// TIA Portal V17 export
// export: Created 2025-03-05T08:00:06.619545Z, ExportSetting WithDefaults, DisplayName Totally Integrated Automation Portal, DisplayVersion V17 Update 8, DisplayName TIA Portal Openness, DisplayVersion V17 Update 8, DisplayName TIA Portal Version Control Interface, DisplayVersion V17, DisplayName SINAMICS Startdrive Advanced, DisplayVersion V17 SP2, DisplayName SINAMICS Startdrive G110M, G120, G120C, G120D, G120P, G115D, DisplayVersion V17 SP2, DisplayName SINAMICS Startdrive G130, G150, S120, S150, SINAMICS MV, S210, DisplayVersion V17 SP2, DisplayName STEP 7 Professional, DisplayVersion V17 Update 8, DisplayName SINUMERIK ONE STEP 7 Toolbox, DisplayVersion V17 Update 12, DisplayName SINUMERIK 840D sl STEP 7 Toolbox, DisplayVersion V17 Update 12, DisplayName STEP 7 Safety, DisplayVersion V17 Update 6, DisplayName WinCC Advanced, DisplayVersion V17 Update 8
FUNCTION "FC2033_RUN_OUT_CYCLE" : Void   // FC2033, LAD
{ S7_Optimized_Access := 'FALSE' }
AUTHOR : ETXETAR
VERSION : 1.0
// stored: AutoNumber false, IsIECCheckEnabled false, SetENOAutomatically false, UDAEnableTagReadback false
   VAR_TEMP
      O_BYTE_0 : Struct   // OPTIONS BYTE 0
         MACH_EMPTY_WITHOUT_STOP_1 : Bool;   // MACHINE EMPTY WITHOUT STOP OPTION
      END_STRUCT;
   END_VAR
   VAR CONSTANT
      FC_NUMBER : DInt := 2033;
   END_VAR
   VAR_TEMP   // added for the SCL form of the ladder/FBD networks
      _w1 : Bool;
      _w2 : Bool;
   END_VAR
BEGIN

REGION Network 1: MACHINE EMPTY WITHOUT STOP OPTION
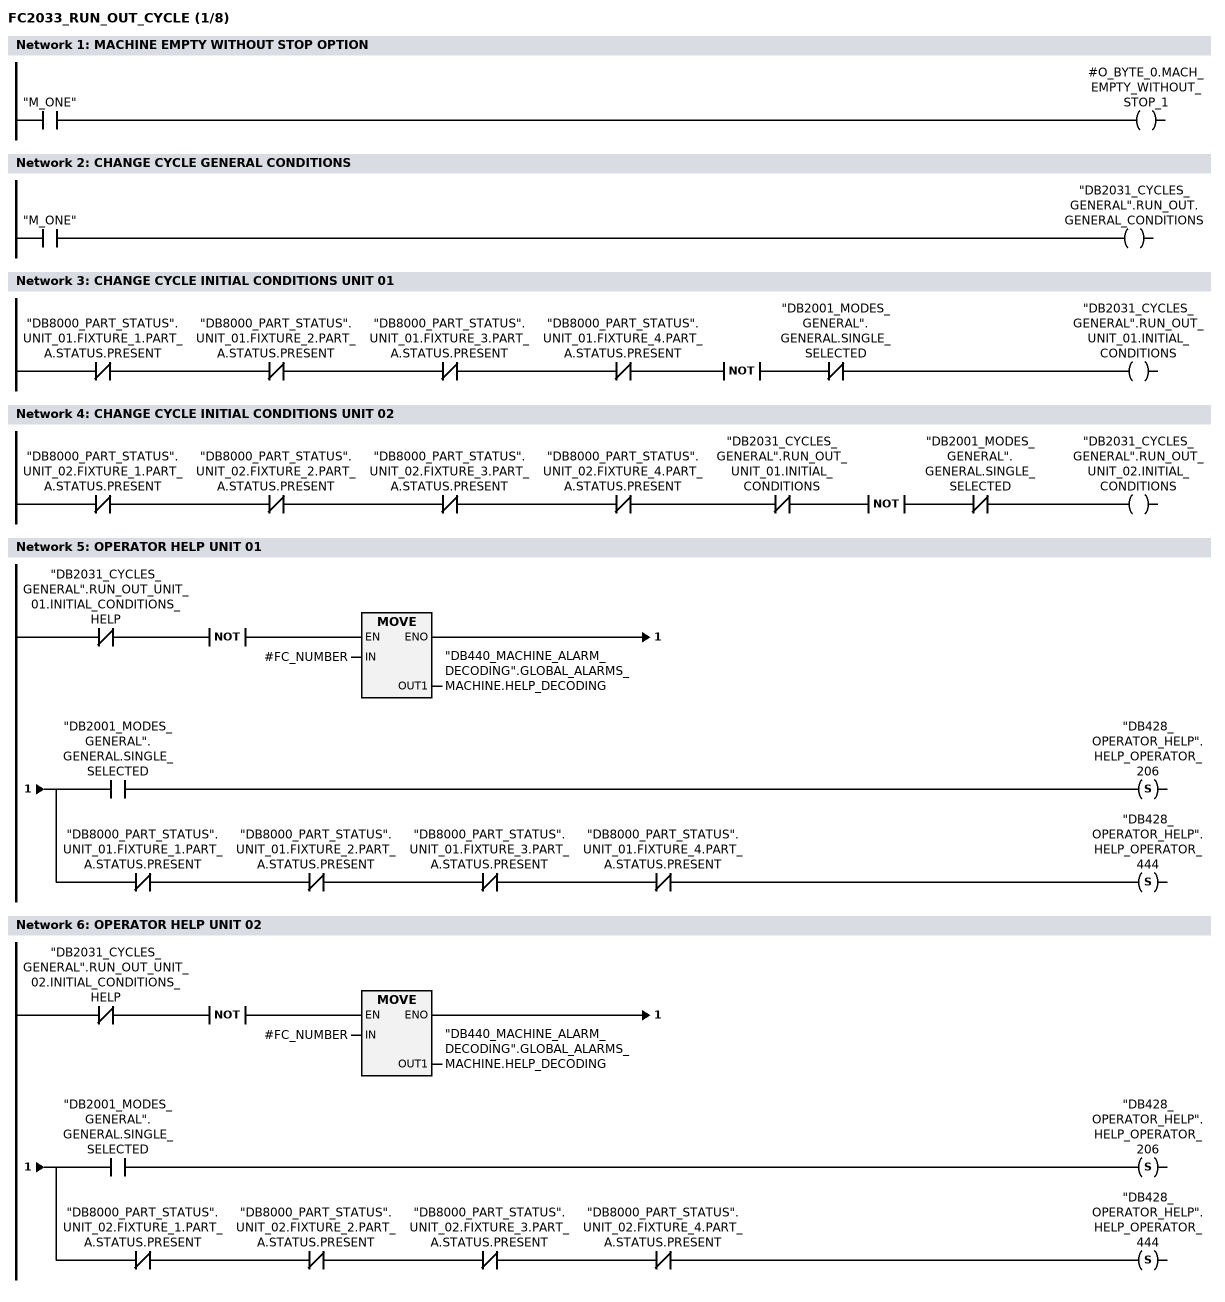
   RUNG wire#powerrail
      Contact( "M_ONE" )
      Coil( #O_BYTE_0.MACH_EMPTY_WITHOUT_STOP_1 )
   END_RUNG
   // the same network as SCL:
   #O_BYTE_0.MACH_EMPTY_WITHOUT_STOP_1 := "M_ONE";
END_REGION

REGION Network 2: CHANGE CYCLE GENERAL CONDITIONS
   RUNG wire#powerrail
      Contact( "M_ONE" )
      Coil( "DB2031_CYCLES_GENERAL".RUN_OUT.GENERAL_CONDITIONS )
   END_RUNG
   // the same network as SCL:
   "DB2031_CYCLES_GENERAL".RUN_OUT.GENERAL_CONDITIONS := "M_ONE";
END_REGION

REGION Network 3: CHANGE CYCLE INITIAL CONDITIONS UNIT 01
   RUNG wire#powerrail
      I_Contact( "DB8000_PART_STATUS".UNIT_01.FIXTURE_1.PART_A.STATUS.PRESENT )
      I_Contact( "DB8000_PART_STATUS".UNIT_01.FIXTURE_2.PART_A.STATUS.PRESENT )
      I_Contact( "DB8000_PART_STATUS".UNIT_01.FIXTURE_3.PART_A.STATUS.PRESENT )
      I_Contact( "DB8000_PART_STATUS".UNIT_01.FIXTURE_4.PART_A.STATUS.PRESENT )
      Not()
      I_Contact( "DB2001_MODES_GENERAL".GENERAL.SINGLE_SELECTED )
      Coil( "DB2031_CYCLES_GENERAL".RUN_OUT_UNIT_01.INITIAL_CONDITIONS )
   END_RUNG
   // the same network as SCL:
   "DB2031_CYCLES_GENERAL".RUN_OUT_UNIT_01.INITIAL_CONDITIONS := NOT (NOT "DB8000_PART_STATUS".UNIT_01.FIXTURE_1.PART_A.STATUS.PRESENT AND NOT "DB8000_PART_STATUS".UNIT_01.FIXTURE_2.PART_A.STATUS.PRESENT AND NOT "DB8000_PART_STATUS".UNIT_01.FIXTURE_3.PART_A.STATUS.PRESENT AND NOT "DB8000_PART_STATUS".UNIT_01.FIXTURE_4.PART_A.STATUS.PRESENT) AND NOT "DB2001_MODES_GENERAL".GENERAL.SINGLE_SELECTED;
END_REGION

REGION Network 4: CHANGE CYCLE INITIAL CONDITIONS UNIT 02
   RUNG wire#powerrail
      I_Contact( "DB8000_PART_STATUS".UNIT_02.FIXTURE_1.PART_A.STATUS.PRESENT )
      I_Contact( "DB8000_PART_STATUS".UNIT_02.FIXTURE_2.PART_A.STATUS.PRESENT )
      I_Contact( "DB8000_PART_STATUS".UNIT_02.FIXTURE_3.PART_A.STATUS.PRESENT )
      I_Contact( "DB8000_PART_STATUS".UNIT_02.FIXTURE_4.PART_A.STATUS.PRESENT )
      I_Contact( "DB2031_CYCLES_GENERAL".RUN_OUT_UNIT_01.INITIAL_CONDITIONS )
      Not()
      I_Contact( "DB2001_MODES_GENERAL".GENERAL.SINGLE_SELECTED )
      Coil( "DB2031_CYCLES_GENERAL".RUN_OUT_UNIT_02.INITIAL_CONDITIONS )
   END_RUNG
   // the same network as SCL:
   "DB2031_CYCLES_GENERAL".RUN_OUT_UNIT_02.INITIAL_CONDITIONS := NOT (NOT "DB8000_PART_STATUS".UNIT_02.FIXTURE_1.PART_A.STATUS.PRESENT AND NOT "DB8000_PART_STATUS".UNIT_02.FIXTURE_2.PART_A.STATUS.PRESENT AND NOT "DB8000_PART_STATUS".UNIT_02.FIXTURE_3.PART_A.STATUS.PRESENT AND NOT "DB8000_PART_STATUS".UNIT_02.FIXTURE_4.PART_A.STATUS.PRESENT AND NOT "DB2031_CYCLES_GENERAL".RUN_OUT_UNIT_01.INITIAL_CONDITIONS) AND NOT "DB2001_MODES_GENERAL".GENERAL.SINGLE_SELECTED;
END_REGION

REGION Network 5: OPERATOR HELP UNIT 01
   RUNG wire#powerrail
      I_Contact( "DB2031_CYCLES_GENERAL".RUN_OUT_UNIT_01.INITIAL_CONDITIONS_HELP )
      Not()
      { S7_GenerateENO := "TRUE" } Move(in := #FC_NUMBER, out1 => "DB440_MACHINE_ALARM_DECODING".GLOBAL_ALARMS_MACHINE.HELP_DECODING)
      wire#w1
      Contact( "DB2001_MODES_GENERAL".GENERAL.SINGLE_SELECTED )
      S_Coil( "DB428_OPERATOR_HELP".HELP_OPERATOR_206 )
   END_RUNG
   RUNG wire#w1
      I_Contact( "DB8000_PART_STATUS".UNIT_01.FIXTURE_1.PART_A.STATUS.PRESENT )
      I_Contact( "DB8000_PART_STATUS".UNIT_01.FIXTURE_2.PART_A.STATUS.PRESENT )
      I_Contact( "DB8000_PART_STATUS".UNIT_01.FIXTURE_3.PART_A.STATUS.PRESENT )
      I_Contact( "DB8000_PART_STATUS".UNIT_01.FIXTURE_4.PART_A.STATUS.PRESENT )
      S_Coil( "DB428_OPERATOR_HELP".HELP_OPERATOR_444 )
   END_RUNG
   // the same network as SCL:
   // ENO of a box is taken as its EN; it also drops when the box reports an error
   #_w1 := NOT (NOT "DB2031_CYCLES_GENERAL".RUN_OUT_UNIT_01.INITIAL_CONDITIONS_HELP);
   IF #_w1 THEN "DB440_MACHINE_ALARM_DECODING".GLOBAL_ALARMS_MACHINE.HELP_DECODING := #FC_NUMBER; END_IF;
   IF #_w1 AND "DB2001_MODES_GENERAL".GENERAL.SINGLE_SELECTED THEN
       "DB428_OPERATOR_HELP".HELP_OPERATOR_206 := TRUE;
   END_IF;
   IF #_w1 AND NOT "DB8000_PART_STATUS".UNIT_01.FIXTURE_1.PART_A.STATUS.PRESENT AND NOT "DB8000_PART_STATUS".UNIT_01.FIXTURE_2.PART_A.STATUS.PRESENT AND NOT "DB8000_PART_STATUS".UNIT_01.FIXTURE_3.PART_A.STATUS.PRESENT AND NOT "DB8000_PART_STATUS".UNIT_01.FIXTURE_4.PART_A.STATUS.PRESENT THEN
       "DB428_OPERATOR_HELP".HELP_OPERATOR_444 := TRUE;
   END_IF;
END_REGION

REGION Network 6: OPERATOR HELP UNIT 02
   RUNG wire#powerrail
      I_Contact( "DB2031_CYCLES_GENERAL".RUN_OUT_UNIT_02.INITIAL_CONDITIONS_HELP )
      Not()
      { S7_GenerateENO := "TRUE" } Move(in := #FC_NUMBER, out1 => "DB440_MACHINE_ALARM_DECODING".GLOBAL_ALARMS_MACHINE.HELP_DECODING)
      wire#w1
      Contact( "DB2001_MODES_GENERAL".GENERAL.SINGLE_SELECTED )
      S_Coil( "DB428_OPERATOR_HELP".HELP_OPERATOR_206 )
   END_RUNG
   RUNG wire#w1
      I_Contact( "DB8000_PART_STATUS".UNIT_02.FIXTURE_1.PART_A.STATUS.PRESENT )
      I_Contact( "DB8000_PART_STATUS".UNIT_02.FIXTURE_2.PART_A.STATUS.PRESENT )
      I_Contact( "DB8000_PART_STATUS".UNIT_02.FIXTURE_3.PART_A.STATUS.PRESENT )
      I_Contact( "DB8000_PART_STATUS".UNIT_02.FIXTURE_4.PART_A.STATUS.PRESENT )
      S_Coil( "DB428_OPERATOR_HELP".HELP_OPERATOR_444 )
   END_RUNG
   // the same network as SCL:
   // ENO of a box is taken as its EN; it also drops when the box reports an error
   #_w1 := NOT (NOT "DB2031_CYCLES_GENERAL".RUN_OUT_UNIT_02.INITIAL_CONDITIONS_HELP);
   IF #_w1 THEN "DB440_MACHINE_ALARM_DECODING".GLOBAL_ALARMS_MACHINE.HELP_DECODING := #FC_NUMBER; END_IF;
   IF #_w1 AND "DB2001_MODES_GENERAL".GENERAL.SINGLE_SELECTED THEN
       "DB428_OPERATOR_HELP".HELP_OPERATOR_206 := TRUE;
   END_IF;
   IF #_w1 AND NOT "DB8000_PART_STATUS".UNIT_02.FIXTURE_1.PART_A.STATUS.PRESENT AND NOT "DB8000_PART_STATUS".UNIT_02.FIXTURE_2.PART_A.STATUS.PRESENT AND NOT "DB8000_PART_STATUS".UNIT_02.FIXTURE_3.PART_A.STATUS.PRESENT AND NOT "DB8000_PART_STATUS".UNIT_02.FIXTURE_4.PART_A.STATUS.PRESENT THEN
       "DB428_OPERATOR_HELP".HELP_OPERATOR_444 := TRUE;
   END_IF;
END_REGION

REGION Network 7: ENABLE REQUEST
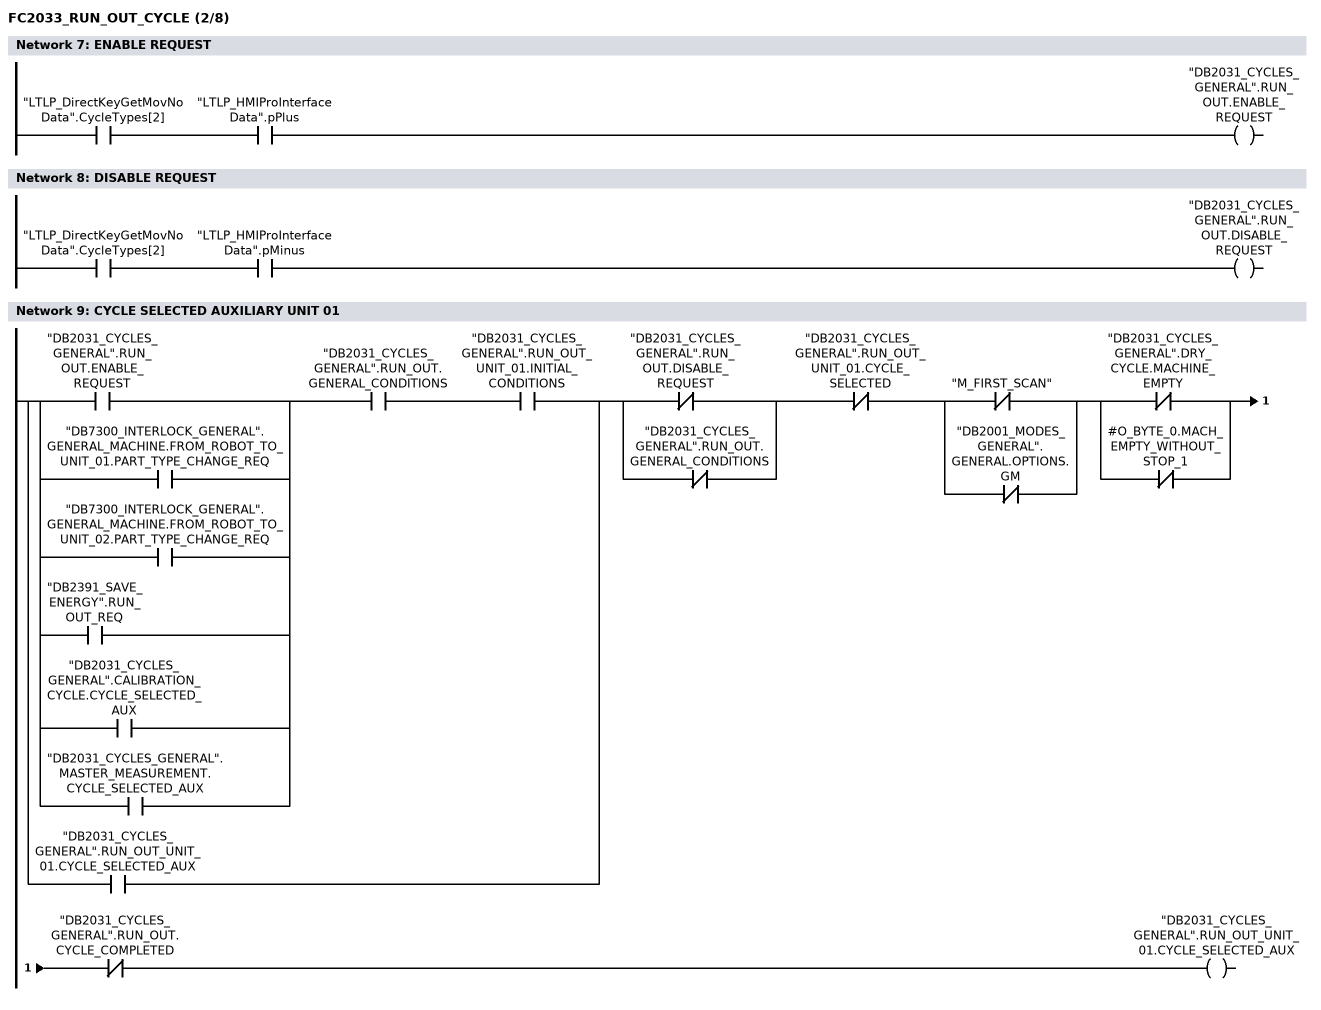
   RUNG wire#powerrail
      Contact( "LTLP_DirectKeyGetMovNoData".CycleTypes[2] )
      Contact( "LTLP_HMIProInterfaceData".pPlus )
      Coil( "DB2031_CYCLES_GENERAL".RUN_OUT.ENABLE_REQUEST )
   END_RUNG
   // the same network as SCL:
   "DB2031_CYCLES_GENERAL".RUN_OUT.ENABLE_REQUEST := "LTLP_DirectKeyGetMovNoData".CycleTypes[2] AND "LTLP_HMIProInterfaceData".pPlus;
END_REGION

REGION Network 8: DISABLE REQUEST
   RUNG wire#powerrail
      Contact( "LTLP_DirectKeyGetMovNoData".CycleTypes[2] )
      Contact( "LTLP_HMIProInterfaceData".pMinus )
      Coil( "DB2031_CYCLES_GENERAL".RUN_OUT.DISABLE_REQUEST )
   END_RUNG
   // the same network as SCL:
   "DB2031_CYCLES_GENERAL".RUN_OUT.DISABLE_REQUEST := "LTLP_DirectKeyGetMovNoData".CycleTypes[2] AND "LTLP_HMIProInterfaceData".pMinus;
END_REGION

REGION Network 9: CYCLE SELECTED AUXILIARY UNIT 01
   RUNG wire#powerrail
      Contact( "DB2031_CYCLES_GENERAL".RUN_OUT.ENABLE_REQUEST )
      wire#w1
      Contact( "DB2031_CYCLES_GENERAL".RUN_OUT.GENERAL_CONDITIONS )
      Contact( "DB2031_CYCLES_GENERAL".RUN_OUT_UNIT_01.INITIAL_CONDITIONS )
      wire#w2
      I_Contact( "DB2031_CYCLES_GENERAL".RUN_OUT.DISABLE_REQUEST )
      wire#w3
      I_Contact( "DB2031_CYCLES_GENERAL".RUN_OUT_UNIT_01.CYCLE_SELECTED )
      wire#w4
      I_Contact( "M_FIRST_SCAN" )
      wire#w5
      I_Contact( "DB2031_CYCLES_GENERAL".DRY_CYCLE.MACHINE_EMPTY )
      wire#w6
      I_Contact( "DB2031_CYCLES_GENERAL".RUN_OUT.CYCLE_COMPLETED )
      Coil( "DB2031_CYCLES_GENERAL".RUN_OUT_UNIT_01.CYCLE_SELECTED_AUX )
   END_RUNG
   RUNG wire#powerrail
      Contact( "DB7300_INTERLOCK_GENERAL".GENERAL_MACHINE.FROM_ROBOT_TO_UNIT_01.PART_TYPE_CHANGE_REQ )
   END_RUNG wire#w1
   RUNG wire#powerrail
      Contact( "DB7300_INTERLOCK_GENERAL".GENERAL_MACHINE.FROM_ROBOT_TO_UNIT_02.PART_TYPE_CHANGE_REQ )
   END_RUNG wire#w1
   RUNG wire#powerrail
      Contact( "DB2391_SAVE_ENERGY".RUN_OUT_REQ )
   END_RUNG wire#w1
   RUNG wire#powerrail
      Contact( "DB2031_CYCLES_GENERAL".CALIBRATION_CYCLE.CYCLE_SELECTED_AUX )
   END_RUNG wire#w1
   RUNG wire#powerrail
      Contact( "DB2031_CYCLES_GENERAL".MASTER_MEASUREMENT.CYCLE_SELECTED_AUX )
   END_RUNG wire#w1
   RUNG wire#powerrail
      Contact( "DB2031_CYCLES_GENERAL".RUN_OUT_UNIT_01.CYCLE_SELECTED_AUX )
   END_RUNG wire#w2
   RUNG wire#w2
      I_Contact( "DB2031_CYCLES_GENERAL".RUN_OUT.GENERAL_CONDITIONS )
   END_RUNG wire#w3
   RUNG wire#w4
      I_Contact( "DB2001_MODES_GENERAL".GENERAL.OPTIONS.GM )
   END_RUNG wire#w5
   RUNG wire#w5
      I_Contact( #O_BYTE_0.MACH_EMPTY_WITHOUT_STOP_1 )
   END_RUNG wire#w6
   // the same network as SCL:
   "DB2031_CYCLES_GENERAL".RUN_OUT_UNIT_01.CYCLE_SELECTED_AUX := ((("DB2031_CYCLES_GENERAL".RUN_OUT.ENABLE_REQUEST OR "DB7300_INTERLOCK_GENERAL".GENERAL_MACHINE.FROM_ROBOT_TO_UNIT_01.PART_TYPE_CHANGE_REQ OR "DB7300_INTERLOCK_GENERAL".GENERAL_MACHINE.FROM_ROBOT_TO_UNIT_02.PART_TYPE_CHANGE_REQ OR "DB2391_SAVE_ENERGY".RUN_OUT_REQ OR "DB2031_CYCLES_GENERAL".CALIBRATION_CYCLE.CYCLE_SELECTED_AUX OR "DB2031_CYCLES_GENERAL".MASTER_MEASUREMENT.CYCLE_SELECTED_AUX) AND "DB2031_CYCLES_GENERAL".RUN_OUT.GENERAL_CONDITIONS AND "DB2031_CYCLES_GENERAL".RUN_OUT_UNIT_01.INITIAL_CONDITIONS) OR "DB2031_CYCLES_GENERAL".RUN_OUT_UNIT_01.CYCLE_SELECTED_AUX) AND (NOT "DB2031_CYCLES_GENERAL".RUN_OUT.DISABLE_REQUEST OR NOT "DB2031_CYCLES_GENERAL".RUN_OUT.GENERAL_CONDITIONS) AND NOT "DB2031_CYCLES_GENERAL".RUN_OUT_UNIT_01.CYCLE_SELECTED AND (NOT "M_FIRST_SCAN" OR NOT "DB2001_MODES_GENERAL".GENERAL.OPTIONS.GM) AND (NOT "DB2031_CYCLES_GENERAL".DRY_CYCLE.MACHINE_EMPTY OR NOT #O_BYTE_0.MACH_EMPTY_WITHOUT_STOP_1) AND NOT "DB2031_CYCLES_GENERAL".RUN_OUT.CYCLE_COMPLETED;
END_REGION

REGION Network 10: CYCLE SELECTED AUXILIARY UNIT 02
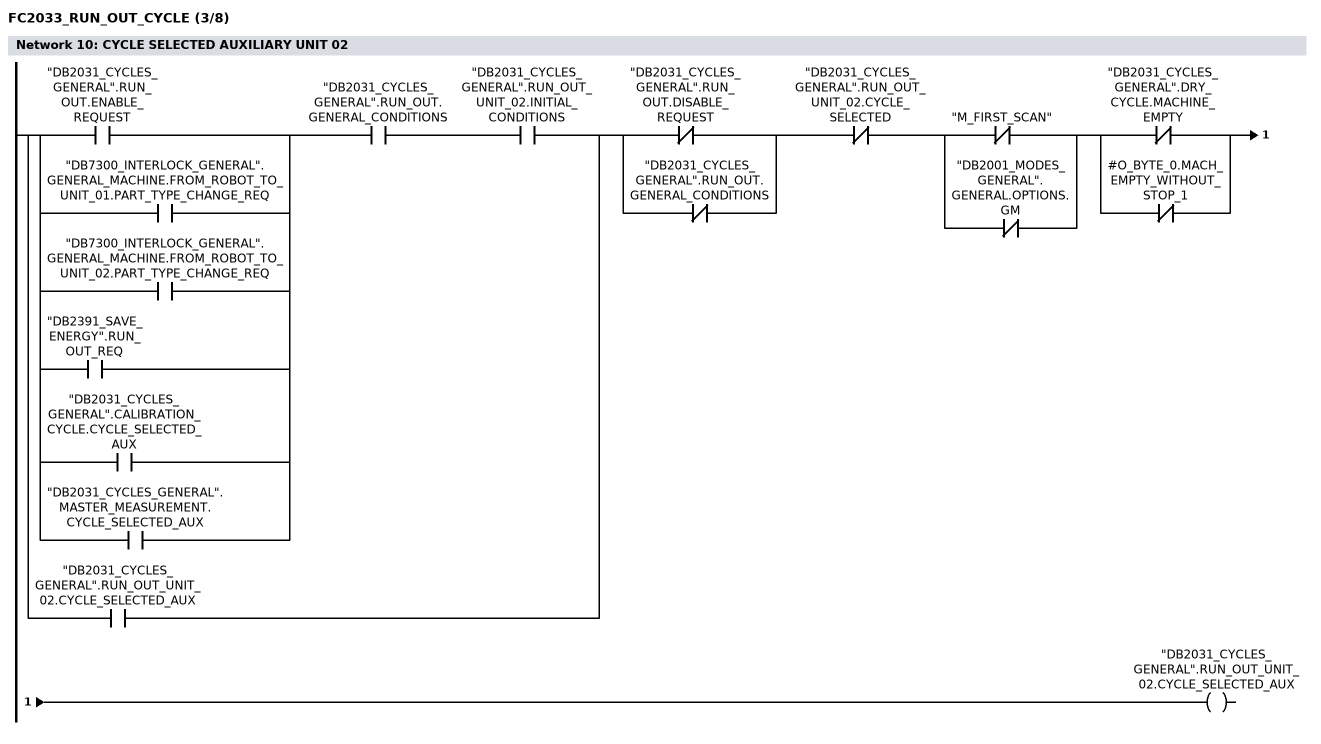
   RUNG wire#powerrail
      Contact( "DB2031_CYCLES_GENERAL".RUN_OUT.ENABLE_REQUEST )
      wire#w1
      Contact( "DB2031_CYCLES_GENERAL".RUN_OUT.GENERAL_CONDITIONS )
      Contact( "DB2031_CYCLES_GENERAL".RUN_OUT_UNIT_02.INITIAL_CONDITIONS )
      wire#w2
      I_Contact( "DB2031_CYCLES_GENERAL".RUN_OUT.DISABLE_REQUEST )
      wire#w3
      I_Contact( "DB2031_CYCLES_GENERAL".RUN_OUT_UNIT_02.CYCLE_SELECTED )
      wire#w4
      I_Contact( "M_FIRST_SCAN" )
      wire#w5
      I_Contact( "DB2031_CYCLES_GENERAL".DRY_CYCLE.MACHINE_EMPTY )
      wire#w6
      Coil( "DB2031_CYCLES_GENERAL".RUN_OUT_UNIT_02.CYCLE_SELECTED_AUX )
   END_RUNG
   RUNG wire#powerrail
      Contact( "DB7300_INTERLOCK_GENERAL".GENERAL_MACHINE.FROM_ROBOT_TO_UNIT_01.PART_TYPE_CHANGE_REQ )
   END_RUNG wire#w1
   RUNG wire#powerrail
      Contact( "DB7300_INTERLOCK_GENERAL".GENERAL_MACHINE.FROM_ROBOT_TO_UNIT_02.PART_TYPE_CHANGE_REQ )
   END_RUNG wire#w1
   RUNG wire#powerrail
      Contact( "DB2391_SAVE_ENERGY".RUN_OUT_REQ )
   END_RUNG wire#w1
   RUNG wire#powerrail
      Contact( "DB2031_CYCLES_GENERAL".CALIBRATION_CYCLE.CYCLE_SELECTED_AUX )
   END_RUNG wire#w1
   RUNG wire#powerrail
      Contact( "DB2031_CYCLES_GENERAL".MASTER_MEASUREMENT.CYCLE_SELECTED_AUX )
   END_RUNG wire#w1
   RUNG wire#powerrail
      Contact( "DB2031_CYCLES_GENERAL".RUN_OUT_UNIT_02.CYCLE_SELECTED_AUX )
   END_RUNG wire#w2
   RUNG wire#w2
      I_Contact( "DB2031_CYCLES_GENERAL".RUN_OUT.GENERAL_CONDITIONS )
   END_RUNG wire#w3
   RUNG wire#w4
      I_Contact( "DB2001_MODES_GENERAL".GENERAL.OPTIONS.GM )
   END_RUNG wire#w5
   RUNG wire#w5
      I_Contact( #O_BYTE_0.MACH_EMPTY_WITHOUT_STOP_1 )
   END_RUNG wire#w6
   // the same network as SCL:
   "DB2031_CYCLES_GENERAL".RUN_OUT_UNIT_02.CYCLE_SELECTED_AUX := ((("DB2031_CYCLES_GENERAL".RUN_OUT.ENABLE_REQUEST OR "DB7300_INTERLOCK_GENERAL".GENERAL_MACHINE.FROM_ROBOT_TO_UNIT_01.PART_TYPE_CHANGE_REQ OR "DB7300_INTERLOCK_GENERAL".GENERAL_MACHINE.FROM_ROBOT_TO_UNIT_02.PART_TYPE_CHANGE_REQ OR "DB2391_SAVE_ENERGY".RUN_OUT_REQ OR "DB2031_CYCLES_GENERAL".CALIBRATION_CYCLE.CYCLE_SELECTED_AUX OR "DB2031_CYCLES_GENERAL".MASTER_MEASUREMENT.CYCLE_SELECTED_AUX) AND "DB2031_CYCLES_GENERAL".RUN_OUT.GENERAL_CONDITIONS AND "DB2031_CYCLES_GENERAL".RUN_OUT_UNIT_02.INITIAL_CONDITIONS) OR "DB2031_CYCLES_GENERAL".RUN_OUT_UNIT_02.CYCLE_SELECTED_AUX) AND (NOT "DB2031_CYCLES_GENERAL".RUN_OUT.DISABLE_REQUEST OR NOT "DB2031_CYCLES_GENERAL".RUN_OUT.GENERAL_CONDITIONS) AND NOT "DB2031_CYCLES_GENERAL".RUN_OUT_UNIT_02.CYCLE_SELECTED AND (NOT "M_FIRST_SCAN" OR NOT "DB2001_MODES_GENERAL".GENERAL.OPTIONS.GM) AND (NOT "DB2031_CYCLES_GENERAL".DRY_CYCLE.MACHINE_EMPTY OR NOT #O_BYTE_0.MACH_EMPTY_WITHOUT_STOP_1);
END_REGION

REGION Network 11: CYCLE SELECTED UNIT 01
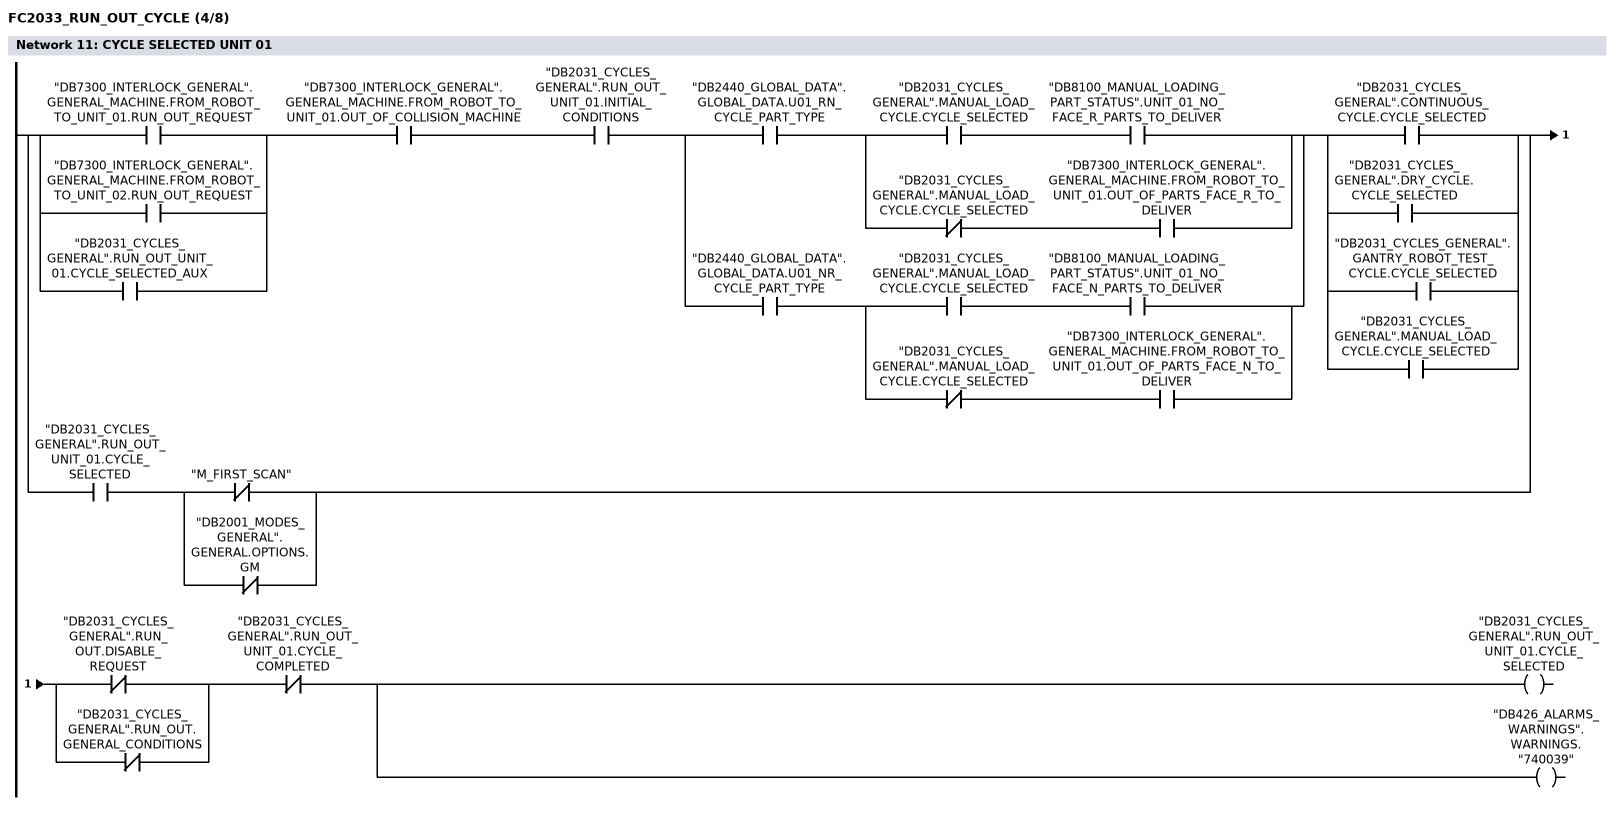
   RUNG wire#powerrail
      Contact( "DB7300_INTERLOCK_GENERAL".GENERAL_MACHINE.FROM_ROBOT_TO_UNIT_01.RUN_OUT_REQUEST )
      wire#w1
      Contact( "DB7300_INTERLOCK_GENERAL".GENERAL_MACHINE.FROM_ROBOT_TO_UNIT_01.OUT_OF_COLLISION_MACHINE )
      Contact( "DB2031_CYCLES_GENERAL".RUN_OUT_UNIT_01.INITIAL_CONDITIONS )
      wire#w2
      Contact( "DB2440_GLOBAL_DATA".GLOBAL_DATA.U01_RN_CYCLE_PART_TYPE )
      wire#w3
      Contact( "DB2031_CYCLES_GENERAL".MANUAL_LOAD_CYCLE.CYCLE_SELECTED )
      Contact( "DB8100_MANUAL_LOADING_PART_STATUS".UNIT_01_NO_FACE_R_PARTS_TO_DELIVER )
      wire#w4
      Contact( "DB2031_CYCLES_GENERAL".CONTINUOUS_CYCLE.CYCLE_SELECTED )
      wire#w6
      I_Contact( "DB2031_CYCLES_GENERAL".RUN_OUT.DISABLE_REQUEST )
      wire#w8
      I_Contact( "DB2031_CYCLES_GENERAL".RUN_OUT_UNIT_01.CYCLE_COMPLETED )
      wire#w9
      Coil( "DB2031_CYCLES_GENERAL".RUN_OUT_UNIT_01.CYCLE_SELECTED )
   END_RUNG
   RUNG wire#powerrail
      Contact( "DB7300_INTERLOCK_GENERAL".GENERAL_MACHINE.FROM_ROBOT_TO_UNIT_02.RUN_OUT_REQUEST )
   END_RUNG wire#w1
   RUNG wire#powerrail
      Contact( "DB2031_CYCLES_GENERAL".RUN_OUT_UNIT_01.CYCLE_SELECTED_AUX )
   END_RUNG wire#w1
   RUNG wire#w3
      I_Contact( "DB2031_CYCLES_GENERAL".MANUAL_LOAD_CYCLE.CYCLE_SELECTED )
      Contact( "DB7300_INTERLOCK_GENERAL".GENERAL_MACHINE.FROM_ROBOT_TO_UNIT_01.OUT_OF_PARTS_FACE_R_TO_DELIVER )
   END_RUNG wire#w4
   RUNG wire#w2
      Contact( "DB2440_GLOBAL_DATA".GLOBAL_DATA.U01_NR_CYCLE_PART_TYPE )
      wire#w5
      Contact( "DB2031_CYCLES_GENERAL".MANUAL_LOAD_CYCLE.CYCLE_SELECTED )
      Contact( "DB8100_MANUAL_LOADING_PART_STATUS".UNIT_01_NO_FACE_N_PARTS_TO_DELIVER )
   END_RUNG wire#w4
   RUNG wire#w5
      I_Contact( "DB2031_CYCLES_GENERAL".MANUAL_LOAD_CYCLE.CYCLE_SELECTED )
      Contact( "DB7300_INTERLOCK_GENERAL".GENERAL_MACHINE.FROM_ROBOT_TO_UNIT_01.OUT_OF_PARTS_FACE_N_TO_DELIVER )
   END_RUNG wire#w4
   RUNG wire#w4
      Contact( "DB2031_CYCLES_GENERAL".DRY_CYCLE.CYCLE_SELECTED )
   END_RUNG wire#w6
   RUNG wire#w4
      Contact( "DB2031_CYCLES_GENERAL".GANTRY_ROBOT_TEST_CYCLE.CYCLE_SELECTED )
   END_RUNG wire#w6
   RUNG wire#w4
      Contact( "DB2031_CYCLES_GENERAL".MANUAL_LOAD_CYCLE.CYCLE_SELECTED )
   END_RUNG wire#w6
   RUNG wire#powerrail
      Contact( "DB2031_CYCLES_GENERAL".RUN_OUT_UNIT_01.CYCLE_SELECTED )
      wire#w7
      I_Contact( "M_FIRST_SCAN" )
   END_RUNG wire#w6
   RUNG wire#w7
      I_Contact( "DB2001_MODES_GENERAL".GENERAL.OPTIONS.GM )
   END_RUNG wire#w6
   RUNG wire#w6
      I_Contact( "DB2031_CYCLES_GENERAL".RUN_OUT.GENERAL_CONDITIONS )
   END_RUNG wire#w8
   RUNG wire#w9
      Coil( "DB426_ALARMS_WARNINGS".WARNINGS."740039" )
   END_RUNG
   // the same network as SCL:
   "DB2031_CYCLES_GENERAL".RUN_OUT_UNIT_01.CYCLE_SELECTED := ((("DB7300_INTERLOCK_GENERAL".GENERAL_MACHINE.FROM_ROBOT_TO_UNIT_01.RUN_OUT_REQUEST OR "DB7300_INTERLOCK_GENERAL".GENERAL_MACHINE.FROM_ROBOT_TO_UNIT_02.RUN_OUT_REQUEST OR "DB2031_CYCLES_GENERAL".RUN_OUT_UNIT_01.CYCLE_SELECTED_AUX) AND "DB7300_INTERLOCK_GENERAL".GENERAL_MACHINE.FROM_ROBOT_TO_UNIT_01.OUT_OF_COLLISION_MACHINE AND "DB2031_CYCLES_GENERAL".RUN_OUT_UNIT_01.INITIAL_CONDITIONS AND (("DB2440_GLOBAL_DATA".GLOBAL_DATA.U01_RN_CYCLE_PART_TYPE AND (("DB2031_CYCLES_GENERAL".MANUAL_LOAD_CYCLE.CYCLE_SELECTED AND "DB8100_MANUAL_LOADING_PART_STATUS".UNIT_01_NO_FACE_R_PARTS_TO_DELIVER) OR (NOT "DB2031_CYCLES_GENERAL".MANUAL_LOAD_CYCLE.CYCLE_SELECTED AND "DB7300_INTERLOCK_GENERAL".GENERAL_MACHINE.FROM_ROBOT_TO_UNIT_01.OUT_OF_PARTS_FACE_R_TO_DELIVER))) OR ("DB2440_GLOBAL_DATA".GLOBAL_DATA.U01_NR_CYCLE_PART_TYPE AND (("DB2031_CYCLES_GENERAL".MANUAL_LOAD_CYCLE.CYCLE_SELECTED AND "DB8100_MANUAL_LOADING_PART_STATUS".UNIT_01_NO_FACE_N_PARTS_TO_DELIVER) OR (NOT "DB2031_CYCLES_GENERAL".MANUAL_LOAD_CYCLE.CYCLE_SELECTED AND "DB7300_INTERLOCK_GENERAL".GENERAL_MACHINE.FROM_ROBOT_TO_UNIT_01.OUT_OF_PARTS_FACE_N_TO_DELIVER)))) AND ("DB2031_CYCLES_GENERAL".CONTINUOUS_CYCLE.CYCLE_SELECTED OR "DB2031_CYCLES_GENERAL".DRY_CYCLE.CYCLE_SELECTED OR "DB2031_CYCLES_GENERAL".GANTRY_ROBOT_TEST_CYCLE.CYCLE_SELECTED OR "DB2031_CYCLES_GENERAL".MANUAL_LOAD_CYCLE.CYCLE_SELECTED)) OR ("DB2031_CYCLES_GENERAL".RUN_OUT_UNIT_01.CYCLE_SELECTED AND (NOT "M_FIRST_SCAN" OR NOT "DB2001_MODES_GENERAL".GENERAL.OPTIONS.GM))) AND (NOT "DB2031_CYCLES_GENERAL".RUN_OUT.DISABLE_REQUEST OR NOT "DB2031_CYCLES_GENERAL".RUN_OUT.GENERAL_CONDITIONS) AND NOT "DB2031_CYCLES_GENERAL".RUN_OUT_UNIT_01.CYCLE_COMPLETED;
   "DB426_ALARMS_WARNINGS".WARNINGS."740039" := "DB2031_CYCLES_GENERAL".RUN_OUT_UNIT_01.CYCLE_SELECTED;
END_REGION

REGION Network 12: CYCLE SELECTED UNIT 02
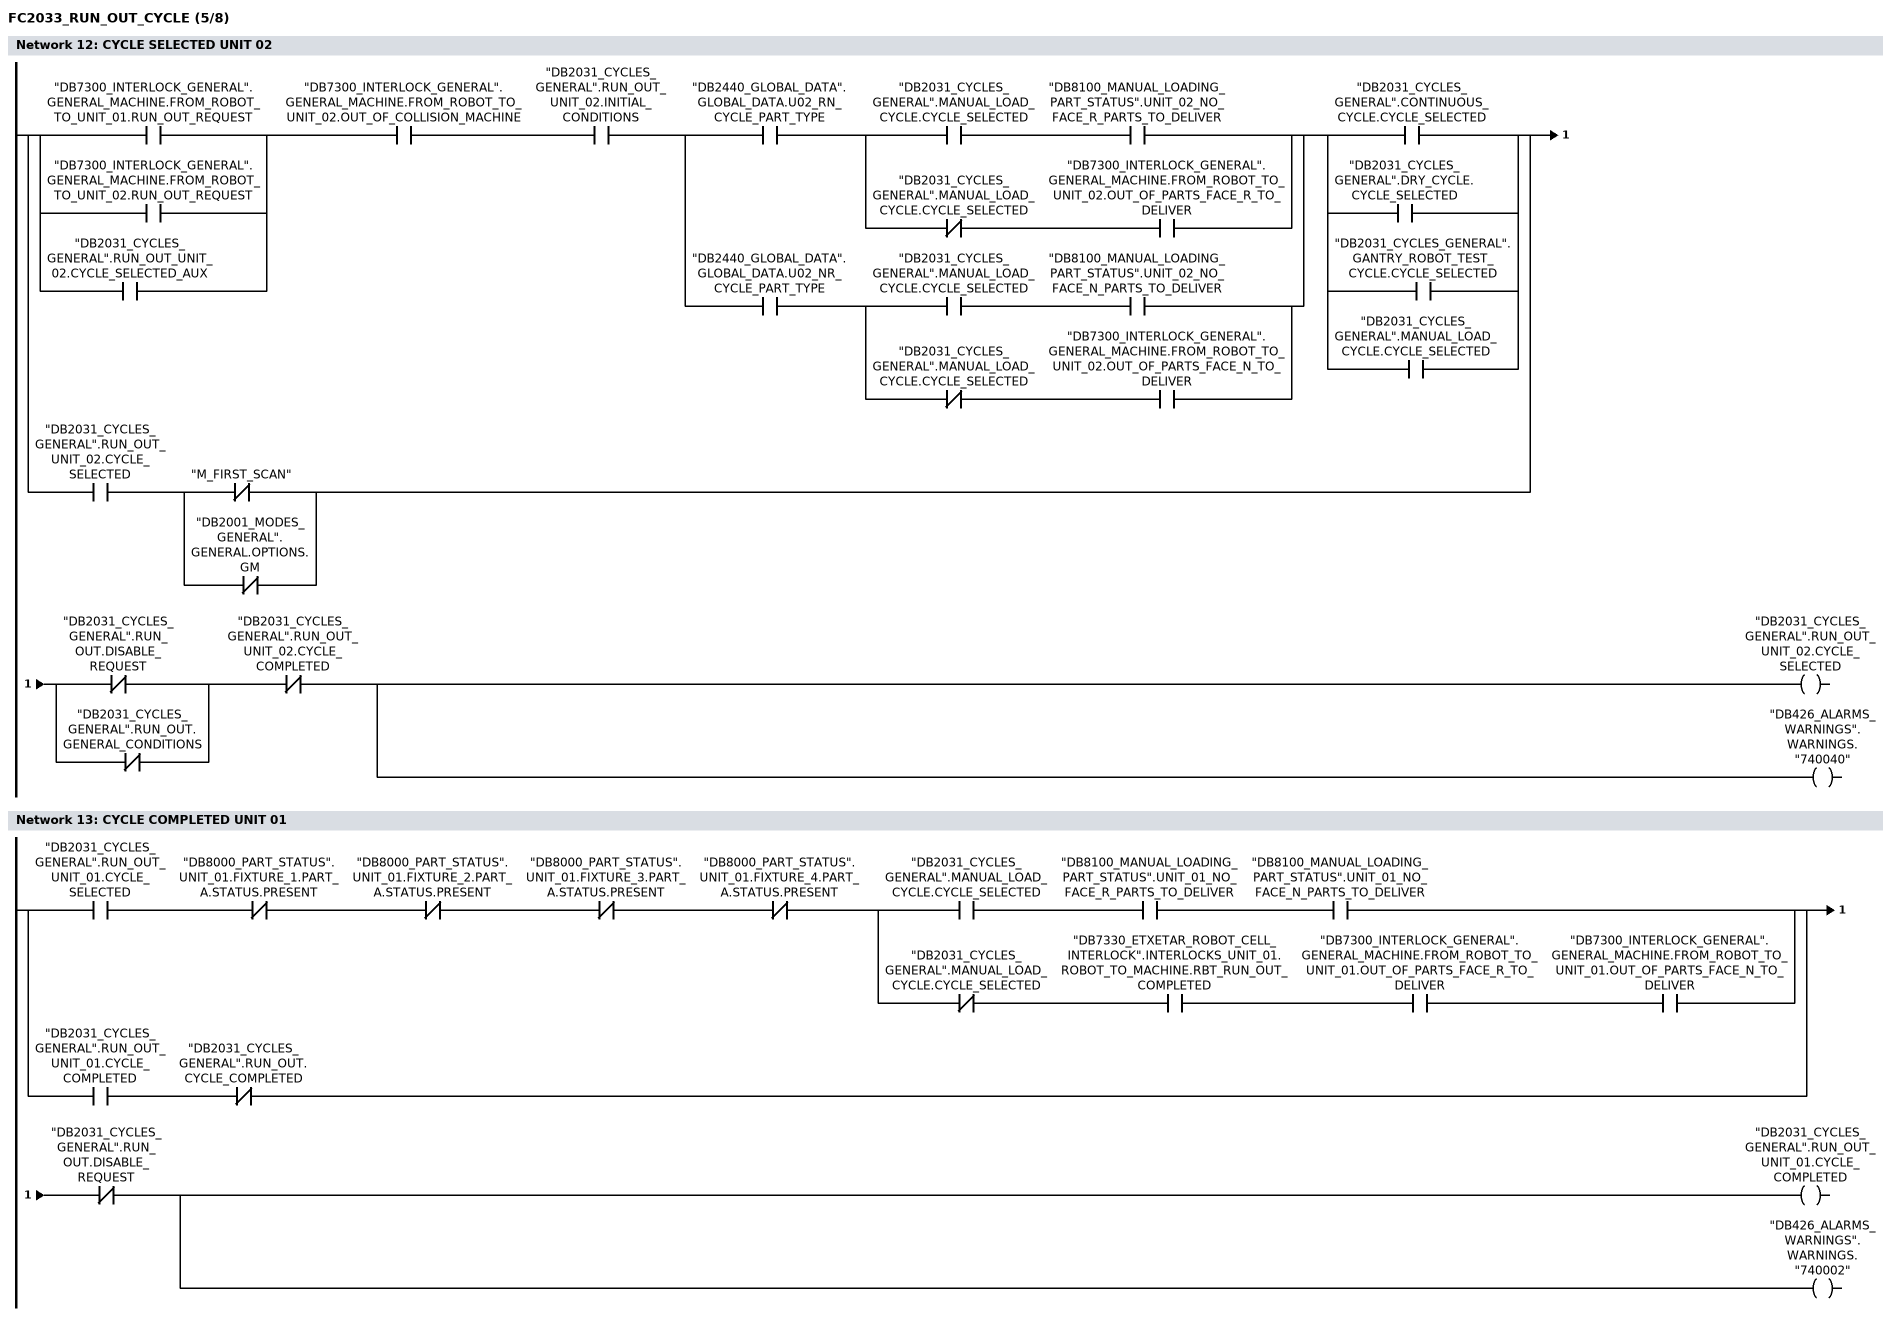
   RUNG wire#powerrail
      Contact( "DB7300_INTERLOCK_GENERAL".GENERAL_MACHINE.FROM_ROBOT_TO_UNIT_01.RUN_OUT_REQUEST )
      wire#w1
      Contact( "DB7300_INTERLOCK_GENERAL".GENERAL_MACHINE.FROM_ROBOT_TO_UNIT_02.OUT_OF_COLLISION_MACHINE )
      Contact( "DB2031_CYCLES_GENERAL".RUN_OUT_UNIT_02.INITIAL_CONDITIONS )
      wire#w2
      Contact( "DB2440_GLOBAL_DATA".GLOBAL_DATA.U02_RN_CYCLE_PART_TYPE )
      wire#w3
      Contact( "DB2031_CYCLES_GENERAL".MANUAL_LOAD_CYCLE.CYCLE_SELECTED )
      Contact( "DB8100_MANUAL_LOADING_PART_STATUS".UNIT_02_NO_FACE_R_PARTS_TO_DELIVER )
      wire#w4
      Contact( "DB2031_CYCLES_GENERAL".CONTINUOUS_CYCLE.CYCLE_SELECTED )
      wire#w6
      I_Contact( "DB2031_CYCLES_GENERAL".RUN_OUT.DISABLE_REQUEST )
      wire#w8
      I_Contact( "DB2031_CYCLES_GENERAL".RUN_OUT_UNIT_02.CYCLE_COMPLETED )
      wire#w9
      Coil( "DB2031_CYCLES_GENERAL".RUN_OUT_UNIT_02.CYCLE_SELECTED )
   END_RUNG
   RUNG wire#powerrail
      Contact( "DB7300_INTERLOCK_GENERAL".GENERAL_MACHINE.FROM_ROBOT_TO_UNIT_02.RUN_OUT_REQUEST )
   END_RUNG wire#w1
   RUNG wire#powerrail
      Contact( "DB2031_CYCLES_GENERAL".RUN_OUT_UNIT_02.CYCLE_SELECTED_AUX )
   END_RUNG wire#w1
   RUNG wire#w3
      I_Contact( "DB2031_CYCLES_GENERAL".MANUAL_LOAD_CYCLE.CYCLE_SELECTED )
      Contact( "DB7300_INTERLOCK_GENERAL".GENERAL_MACHINE.FROM_ROBOT_TO_UNIT_02.OUT_OF_PARTS_FACE_R_TO_DELIVER )
   END_RUNG wire#w4
   RUNG wire#w2
      Contact( "DB2440_GLOBAL_DATA".GLOBAL_DATA.U02_NR_CYCLE_PART_TYPE )
      wire#w5
      Contact( "DB2031_CYCLES_GENERAL".MANUAL_LOAD_CYCLE.CYCLE_SELECTED )
      Contact( "DB8100_MANUAL_LOADING_PART_STATUS".UNIT_02_NO_FACE_N_PARTS_TO_DELIVER )
   END_RUNG wire#w4
   RUNG wire#w5
      I_Contact( "DB2031_CYCLES_GENERAL".MANUAL_LOAD_CYCLE.CYCLE_SELECTED )
      Contact( "DB7300_INTERLOCK_GENERAL".GENERAL_MACHINE.FROM_ROBOT_TO_UNIT_02.OUT_OF_PARTS_FACE_N_TO_DELIVER )
   END_RUNG wire#w4
   RUNG wire#w4
      Contact( "DB2031_CYCLES_GENERAL".DRY_CYCLE.CYCLE_SELECTED )
   END_RUNG wire#w6
   RUNG wire#w4
      Contact( "DB2031_CYCLES_GENERAL".GANTRY_ROBOT_TEST_CYCLE.CYCLE_SELECTED )
   END_RUNG wire#w6
   RUNG wire#w4
      Contact( "DB2031_CYCLES_GENERAL".MANUAL_LOAD_CYCLE.CYCLE_SELECTED )
   END_RUNG wire#w6
   RUNG wire#powerrail
      Contact( "DB2031_CYCLES_GENERAL".RUN_OUT_UNIT_02.CYCLE_SELECTED )
      wire#w7
      I_Contact( "M_FIRST_SCAN" )
   END_RUNG wire#w6
   RUNG wire#w7
      I_Contact( "DB2001_MODES_GENERAL".GENERAL.OPTIONS.GM )
   END_RUNG wire#w6
   RUNG wire#w6
      I_Contact( "DB2031_CYCLES_GENERAL".RUN_OUT.GENERAL_CONDITIONS )
   END_RUNG wire#w8
   RUNG wire#w9
      Coil( "DB426_ALARMS_WARNINGS".WARNINGS."740040" )
   END_RUNG
   // the same network as SCL:
   "DB2031_CYCLES_GENERAL".RUN_OUT_UNIT_02.CYCLE_SELECTED := ((("DB7300_INTERLOCK_GENERAL".GENERAL_MACHINE.FROM_ROBOT_TO_UNIT_01.RUN_OUT_REQUEST OR "DB7300_INTERLOCK_GENERAL".GENERAL_MACHINE.FROM_ROBOT_TO_UNIT_02.RUN_OUT_REQUEST OR "DB2031_CYCLES_GENERAL".RUN_OUT_UNIT_02.CYCLE_SELECTED_AUX) AND "DB7300_INTERLOCK_GENERAL".GENERAL_MACHINE.FROM_ROBOT_TO_UNIT_02.OUT_OF_COLLISION_MACHINE AND "DB2031_CYCLES_GENERAL".RUN_OUT_UNIT_02.INITIAL_CONDITIONS AND (("DB2440_GLOBAL_DATA".GLOBAL_DATA.U02_RN_CYCLE_PART_TYPE AND (("DB2031_CYCLES_GENERAL".MANUAL_LOAD_CYCLE.CYCLE_SELECTED AND "DB8100_MANUAL_LOADING_PART_STATUS".UNIT_02_NO_FACE_R_PARTS_TO_DELIVER) OR (NOT "DB2031_CYCLES_GENERAL".MANUAL_LOAD_CYCLE.CYCLE_SELECTED AND "DB7300_INTERLOCK_GENERAL".GENERAL_MACHINE.FROM_ROBOT_TO_UNIT_02.OUT_OF_PARTS_FACE_R_TO_DELIVER))) OR ("DB2440_GLOBAL_DATA".GLOBAL_DATA.U02_NR_CYCLE_PART_TYPE AND (("DB2031_CYCLES_GENERAL".MANUAL_LOAD_CYCLE.CYCLE_SELECTED AND "DB8100_MANUAL_LOADING_PART_STATUS".UNIT_02_NO_FACE_N_PARTS_TO_DELIVER) OR (NOT "DB2031_CYCLES_GENERAL".MANUAL_LOAD_CYCLE.CYCLE_SELECTED AND "DB7300_INTERLOCK_GENERAL".GENERAL_MACHINE.FROM_ROBOT_TO_UNIT_02.OUT_OF_PARTS_FACE_N_TO_DELIVER)))) AND ("DB2031_CYCLES_GENERAL".CONTINUOUS_CYCLE.CYCLE_SELECTED OR "DB2031_CYCLES_GENERAL".DRY_CYCLE.CYCLE_SELECTED OR "DB2031_CYCLES_GENERAL".GANTRY_ROBOT_TEST_CYCLE.CYCLE_SELECTED OR "DB2031_CYCLES_GENERAL".MANUAL_LOAD_CYCLE.CYCLE_SELECTED)) OR ("DB2031_CYCLES_GENERAL".RUN_OUT_UNIT_02.CYCLE_SELECTED AND (NOT "M_FIRST_SCAN" OR NOT "DB2001_MODES_GENERAL".GENERAL.OPTIONS.GM))) AND (NOT "DB2031_CYCLES_GENERAL".RUN_OUT.DISABLE_REQUEST OR NOT "DB2031_CYCLES_GENERAL".RUN_OUT.GENERAL_CONDITIONS) AND NOT "DB2031_CYCLES_GENERAL".RUN_OUT_UNIT_02.CYCLE_COMPLETED;
   "DB426_ALARMS_WARNINGS".WARNINGS."740040" := "DB2031_CYCLES_GENERAL".RUN_OUT_UNIT_02.CYCLE_SELECTED;
END_REGION

REGION Network 13: CYCLE COMPLETED UNIT 01
   RUNG wire#powerrail
      Contact( "DB2031_CYCLES_GENERAL".RUN_OUT_UNIT_01.CYCLE_SELECTED )
      I_Contact( "DB8000_PART_STATUS".UNIT_01.FIXTURE_1.PART_A.STATUS.PRESENT )
      I_Contact( "DB8000_PART_STATUS".UNIT_01.FIXTURE_2.PART_A.STATUS.PRESENT )
      I_Contact( "DB8000_PART_STATUS".UNIT_01.FIXTURE_3.PART_A.STATUS.PRESENT )
      I_Contact( "DB8000_PART_STATUS".UNIT_01.FIXTURE_4.PART_A.STATUS.PRESENT )
      wire#w1
      Contact( "DB2031_CYCLES_GENERAL".MANUAL_LOAD_CYCLE.CYCLE_SELECTED )
      Contact( "DB8100_MANUAL_LOADING_PART_STATUS".UNIT_01_NO_FACE_R_PARTS_TO_DELIVER )
      Contact( "DB8100_MANUAL_LOADING_PART_STATUS".UNIT_01_NO_FACE_N_PARTS_TO_DELIVER )
      wire#w2
      I_Contact( "DB2031_CYCLES_GENERAL".RUN_OUT.DISABLE_REQUEST )
      wire#w3
      Coil( "DB2031_CYCLES_GENERAL".RUN_OUT_UNIT_01.CYCLE_COMPLETED )
   END_RUNG
   RUNG wire#w1
      I_Contact( "DB2031_CYCLES_GENERAL".MANUAL_LOAD_CYCLE.CYCLE_SELECTED )
      Contact( "DB7330_ETXETAR_ROBOT_CELL_INTERLOCK".INTERLOCKS_UNIT_01.ROBOT_TO_MACHINE.RBT_RUN_OUT_COMPLETED )
      Contact( "DB7300_INTERLOCK_GENERAL".GENERAL_MACHINE.FROM_ROBOT_TO_UNIT_01.OUT_OF_PARTS_FACE_R_TO_DELIVER )
      Contact( "DB7300_INTERLOCK_GENERAL".GENERAL_MACHINE.FROM_ROBOT_TO_UNIT_01.OUT_OF_PARTS_FACE_N_TO_DELIVER )
   END_RUNG wire#w2
   RUNG wire#powerrail
      Contact( "DB2031_CYCLES_GENERAL".RUN_OUT_UNIT_01.CYCLE_COMPLETED )
      I_Contact( "DB2031_CYCLES_GENERAL".RUN_OUT.CYCLE_COMPLETED )
   END_RUNG wire#w2
   RUNG wire#w3
      Coil( "DB426_ALARMS_WARNINGS".WARNINGS."740002" )
   END_RUNG
   // the same network as SCL:
   "DB2031_CYCLES_GENERAL".RUN_OUT_UNIT_01.CYCLE_COMPLETED := (("DB2031_CYCLES_GENERAL".RUN_OUT_UNIT_01.CYCLE_SELECTED AND NOT "DB8000_PART_STATUS".UNIT_01.FIXTURE_1.PART_A.STATUS.PRESENT AND NOT "DB8000_PART_STATUS".UNIT_01.FIXTURE_2.PART_A.STATUS.PRESENT AND NOT "DB8000_PART_STATUS".UNIT_01.FIXTURE_3.PART_A.STATUS.PRESENT AND NOT "DB8000_PART_STATUS".UNIT_01.FIXTURE_4.PART_A.STATUS.PRESENT AND (("DB2031_CYCLES_GENERAL".MANUAL_LOAD_CYCLE.CYCLE_SELECTED AND "DB8100_MANUAL_LOADING_PART_STATUS".UNIT_01_NO_FACE_R_PARTS_TO_DELIVER AND "DB8100_MANUAL_LOADING_PART_STATUS".UNIT_01_NO_FACE_N_PARTS_TO_DELIVER) OR (NOT "DB2031_CYCLES_GENERAL".MANUAL_LOAD_CYCLE.CYCLE_SELECTED AND "DB7330_ETXETAR_ROBOT_CELL_INTERLOCK".INTERLOCKS_UNIT_01.ROBOT_TO_MACHINE.RBT_RUN_OUT_COMPLETED AND "DB7300_INTERLOCK_GENERAL".GENERAL_MACHINE.FROM_ROBOT_TO_UNIT_01.OUT_OF_PARTS_FACE_R_TO_DELIVER AND "DB7300_INTERLOCK_GENERAL".GENERAL_MACHINE.FROM_ROBOT_TO_UNIT_01.OUT_OF_PARTS_FACE_N_TO_DELIVER))) OR ("DB2031_CYCLES_GENERAL".RUN_OUT_UNIT_01.CYCLE_COMPLETED AND NOT "DB2031_CYCLES_GENERAL".RUN_OUT.CYCLE_COMPLETED)) AND NOT "DB2031_CYCLES_GENERAL".RUN_OUT.DISABLE_REQUEST;
   "DB426_ALARMS_WARNINGS".WARNINGS."740002" := "DB2031_CYCLES_GENERAL".RUN_OUT_UNIT_01.CYCLE_COMPLETED;
END_REGION

REGION Network 14: CYCLE COMPLETED UNIT 02
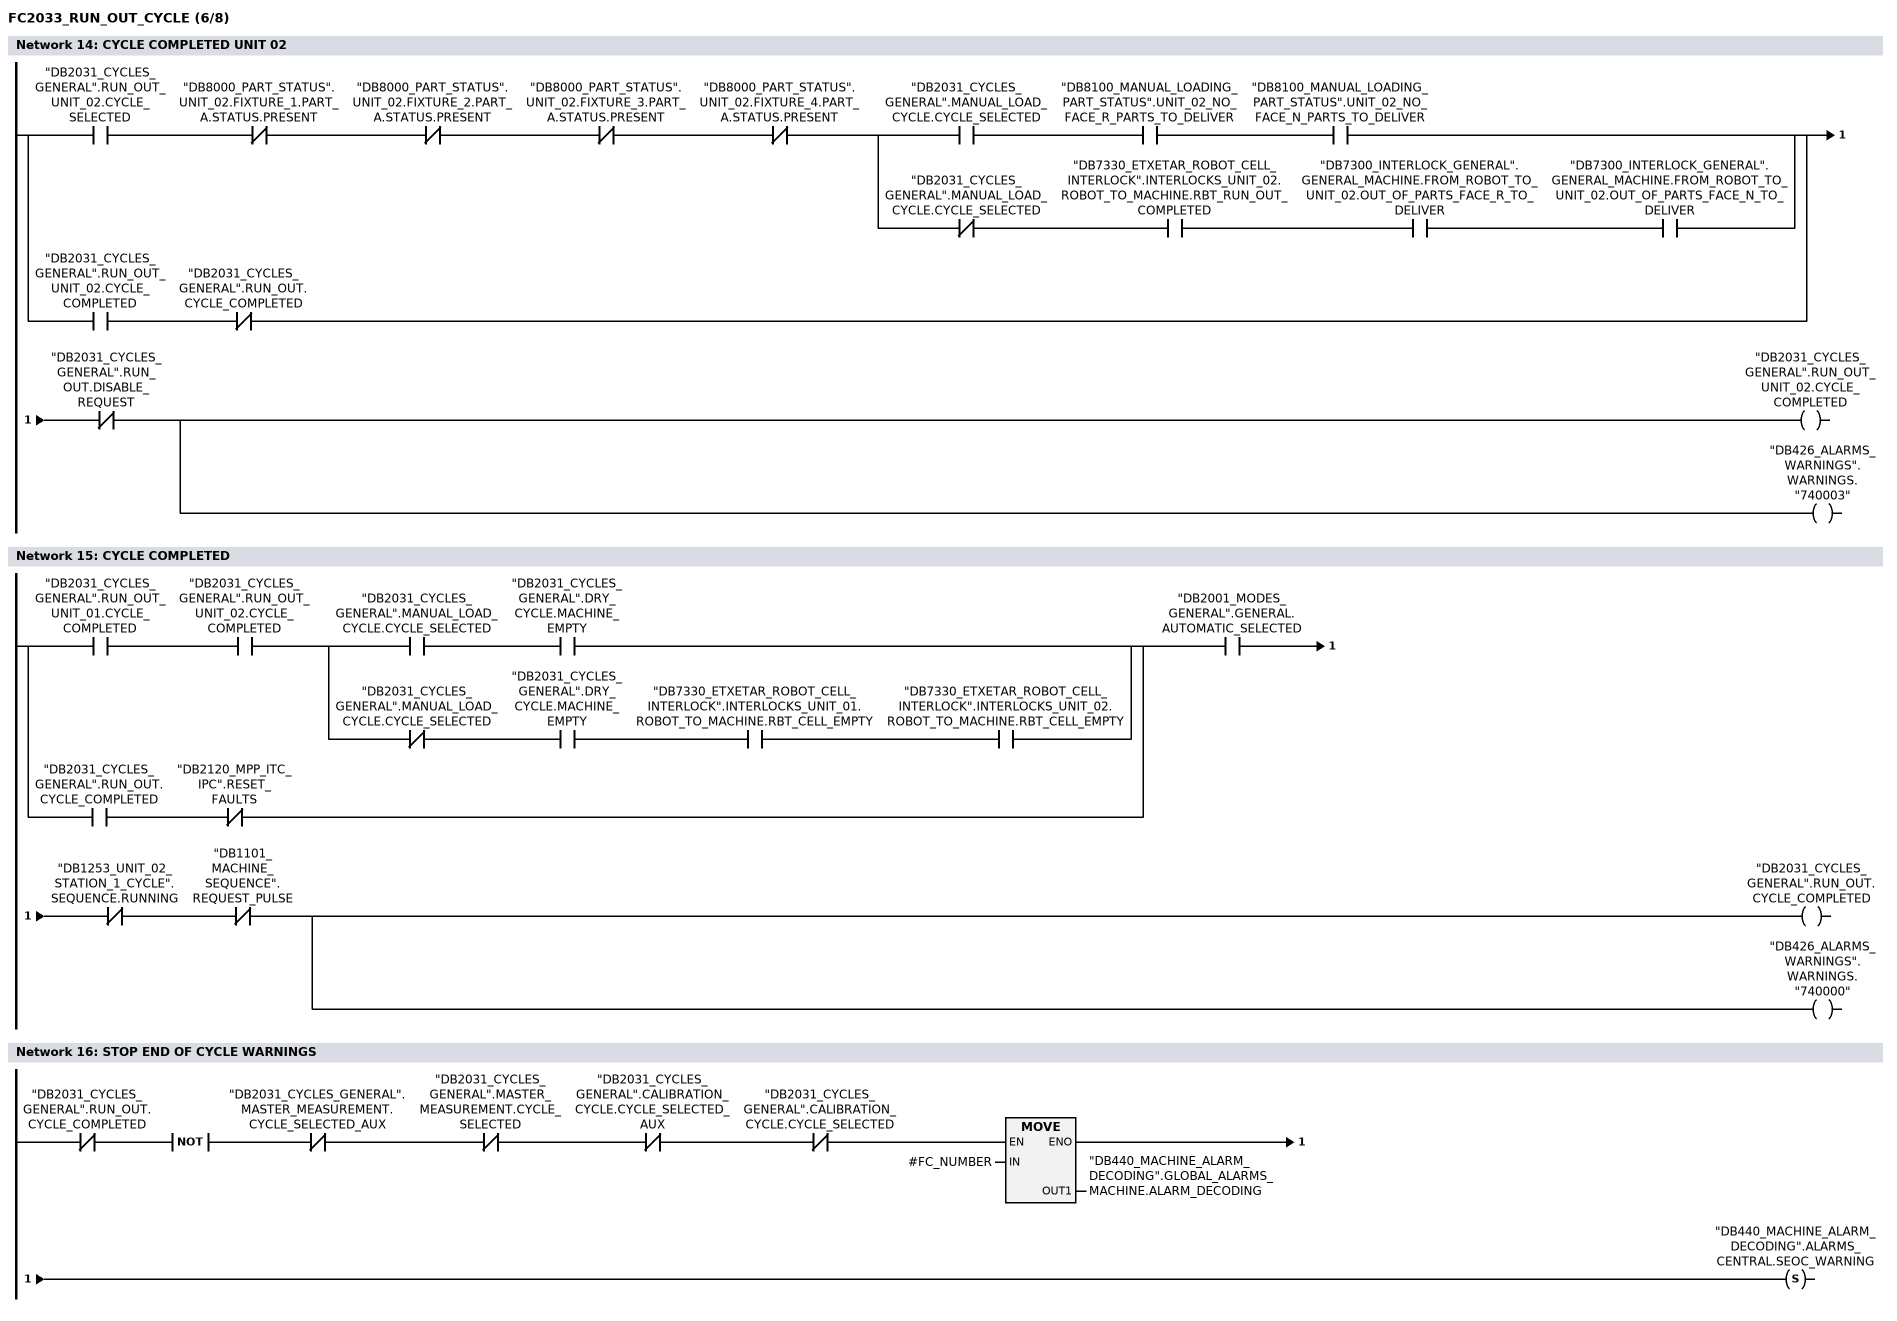
   RUNG wire#powerrail
      Contact( "DB2031_CYCLES_GENERAL".RUN_OUT_UNIT_02.CYCLE_SELECTED )
      I_Contact( "DB8000_PART_STATUS".UNIT_02.FIXTURE_1.PART_A.STATUS.PRESENT )
      I_Contact( "DB8000_PART_STATUS".UNIT_02.FIXTURE_2.PART_A.STATUS.PRESENT )
      I_Contact( "DB8000_PART_STATUS".UNIT_02.FIXTURE_3.PART_A.STATUS.PRESENT )
      I_Contact( "DB8000_PART_STATUS".UNIT_02.FIXTURE_4.PART_A.STATUS.PRESENT )
      wire#w1
      Contact( "DB2031_CYCLES_GENERAL".MANUAL_LOAD_CYCLE.CYCLE_SELECTED )
      Contact( "DB8100_MANUAL_LOADING_PART_STATUS".UNIT_02_NO_FACE_R_PARTS_TO_DELIVER )
      Contact( "DB8100_MANUAL_LOADING_PART_STATUS".UNIT_02_NO_FACE_N_PARTS_TO_DELIVER )
      wire#w2
      I_Contact( "DB2031_CYCLES_GENERAL".RUN_OUT.DISABLE_REQUEST )
      wire#w3
      Coil( "DB2031_CYCLES_GENERAL".RUN_OUT_UNIT_02.CYCLE_COMPLETED )
   END_RUNG
   RUNG wire#w1
      I_Contact( "DB2031_CYCLES_GENERAL".MANUAL_LOAD_CYCLE.CYCLE_SELECTED )
      Contact( "DB7330_ETXETAR_ROBOT_CELL_INTERLOCK".INTERLOCKS_UNIT_02.ROBOT_TO_MACHINE.RBT_RUN_OUT_COMPLETED )
      Contact( "DB7300_INTERLOCK_GENERAL".GENERAL_MACHINE.FROM_ROBOT_TO_UNIT_02.OUT_OF_PARTS_FACE_R_TO_DELIVER )
      Contact( "DB7300_INTERLOCK_GENERAL".GENERAL_MACHINE.FROM_ROBOT_TO_UNIT_02.OUT_OF_PARTS_FACE_N_TO_DELIVER )
   END_RUNG wire#w2
   RUNG wire#powerrail
      Contact( "DB2031_CYCLES_GENERAL".RUN_OUT_UNIT_02.CYCLE_COMPLETED )
      I_Contact( "DB2031_CYCLES_GENERAL".RUN_OUT.CYCLE_COMPLETED )
   END_RUNG wire#w2
   RUNG wire#w3
      Coil( "DB426_ALARMS_WARNINGS".WARNINGS."740003" )
   END_RUNG
   // the same network as SCL:
   "DB2031_CYCLES_GENERAL".RUN_OUT_UNIT_02.CYCLE_COMPLETED := (("DB2031_CYCLES_GENERAL".RUN_OUT_UNIT_02.CYCLE_SELECTED AND NOT "DB8000_PART_STATUS".UNIT_02.FIXTURE_1.PART_A.STATUS.PRESENT AND NOT "DB8000_PART_STATUS".UNIT_02.FIXTURE_2.PART_A.STATUS.PRESENT AND NOT "DB8000_PART_STATUS".UNIT_02.FIXTURE_3.PART_A.STATUS.PRESENT AND NOT "DB8000_PART_STATUS".UNIT_02.FIXTURE_4.PART_A.STATUS.PRESENT AND (("DB2031_CYCLES_GENERAL".MANUAL_LOAD_CYCLE.CYCLE_SELECTED AND "DB8100_MANUAL_LOADING_PART_STATUS".UNIT_02_NO_FACE_R_PARTS_TO_DELIVER AND "DB8100_MANUAL_LOADING_PART_STATUS".UNIT_02_NO_FACE_N_PARTS_TO_DELIVER) OR (NOT "DB2031_CYCLES_GENERAL".MANUAL_LOAD_CYCLE.CYCLE_SELECTED AND "DB7330_ETXETAR_ROBOT_CELL_INTERLOCK".INTERLOCKS_UNIT_02.ROBOT_TO_MACHINE.RBT_RUN_OUT_COMPLETED AND "DB7300_INTERLOCK_GENERAL".GENERAL_MACHINE.FROM_ROBOT_TO_UNIT_02.OUT_OF_PARTS_FACE_R_TO_DELIVER AND "DB7300_INTERLOCK_GENERAL".GENERAL_MACHINE.FROM_ROBOT_TO_UNIT_02.OUT_OF_PARTS_FACE_N_TO_DELIVER))) OR ("DB2031_CYCLES_GENERAL".RUN_OUT_UNIT_02.CYCLE_COMPLETED AND NOT "DB2031_CYCLES_GENERAL".RUN_OUT.CYCLE_COMPLETED)) AND NOT "DB2031_CYCLES_GENERAL".RUN_OUT.DISABLE_REQUEST;
   "DB426_ALARMS_WARNINGS".WARNINGS."740003" := "DB2031_CYCLES_GENERAL".RUN_OUT_UNIT_02.CYCLE_COMPLETED;
END_REGION

REGION Network 15: CYCLE COMPLETED
   RUNG wire#powerrail
      Contact( "DB2031_CYCLES_GENERAL".RUN_OUT_UNIT_01.CYCLE_COMPLETED )
      Contact( "DB2031_CYCLES_GENERAL".RUN_OUT_UNIT_02.CYCLE_COMPLETED )
      wire#w1
      Contact( "DB2031_CYCLES_GENERAL".MANUAL_LOAD_CYCLE.CYCLE_SELECTED )
      Contact( "DB2031_CYCLES_GENERAL".DRY_CYCLE.MACHINE_EMPTY )
      wire#w2
      Contact( "DB2001_MODES_GENERAL".GENERAL.AUTOMATIC_SELECTED )
      I_Contact( "DB1253_UNIT_02_STATION_1_CYCLE".SEQUENCE.RUNNING )
      I_Contact( "DB1101_MACHINE_SEQUENCE".REQUEST_PULSE )
      wire#w3
      Coil( "DB2031_CYCLES_GENERAL".RUN_OUT.CYCLE_COMPLETED )
   END_RUNG
   RUNG wire#w1
      I_Contact( "DB2031_CYCLES_GENERAL".MANUAL_LOAD_CYCLE.CYCLE_SELECTED )
      Contact( "DB2031_CYCLES_GENERAL".DRY_CYCLE.MACHINE_EMPTY )
      Contact( "DB7330_ETXETAR_ROBOT_CELL_INTERLOCK".INTERLOCKS_UNIT_01.ROBOT_TO_MACHINE.RBT_CELL_EMPTY )
      Contact( "DB7330_ETXETAR_ROBOT_CELL_INTERLOCK".INTERLOCKS_UNIT_02.ROBOT_TO_MACHINE.RBT_CELL_EMPTY )
   END_RUNG wire#w2
   RUNG wire#powerrail
      Contact( "DB2031_CYCLES_GENERAL".RUN_OUT.CYCLE_COMPLETED )
      I_Contact( "DB2120_MPP_ITC_IPC".RESET_FAULTS )
   END_RUNG wire#w2
   RUNG wire#w3
      Coil( "DB426_ALARMS_WARNINGS".WARNINGS."740000" )
   END_RUNG
   // the same network as SCL:
   "DB2031_CYCLES_GENERAL".RUN_OUT.CYCLE_COMPLETED := (("DB2031_CYCLES_GENERAL".RUN_OUT_UNIT_01.CYCLE_COMPLETED AND "DB2031_CYCLES_GENERAL".RUN_OUT_UNIT_02.CYCLE_COMPLETED AND (("DB2031_CYCLES_GENERAL".MANUAL_LOAD_CYCLE.CYCLE_SELECTED AND "DB2031_CYCLES_GENERAL".DRY_CYCLE.MACHINE_EMPTY) OR (NOT "DB2031_CYCLES_GENERAL".MANUAL_LOAD_CYCLE.CYCLE_SELECTED AND "DB2031_CYCLES_GENERAL".DRY_CYCLE.MACHINE_EMPTY AND "DB7330_ETXETAR_ROBOT_CELL_INTERLOCK".INTERLOCKS_UNIT_01.ROBOT_TO_MACHINE.RBT_CELL_EMPTY AND "DB7330_ETXETAR_ROBOT_CELL_INTERLOCK".INTERLOCKS_UNIT_02.ROBOT_TO_MACHINE.RBT_CELL_EMPTY))) OR ("DB2031_CYCLES_GENERAL".RUN_OUT.CYCLE_COMPLETED AND NOT "DB2120_MPP_ITC_IPC".RESET_FAULTS)) AND "DB2001_MODES_GENERAL".GENERAL.AUTOMATIC_SELECTED AND NOT "DB1253_UNIT_02_STATION_1_CYCLE".SEQUENCE.RUNNING AND NOT "DB1101_MACHINE_SEQUENCE".REQUEST_PULSE;
   "DB426_ALARMS_WARNINGS".WARNINGS."740000" := "DB2031_CYCLES_GENERAL".RUN_OUT.CYCLE_COMPLETED;
END_REGION

REGION Network 16: STOP END OF CYCLE WARNINGS
   RUNG wire#powerrail
      I_Contact( "DB2031_CYCLES_GENERAL".RUN_OUT.CYCLE_COMPLETED )
      Not()
      I_Contact( "DB2031_CYCLES_GENERAL".MASTER_MEASUREMENT.CYCLE_SELECTED_AUX )
      I_Contact( "DB2031_CYCLES_GENERAL".MASTER_MEASUREMENT.CYCLE_SELECTED )
      I_Contact( "DB2031_CYCLES_GENERAL".CALIBRATION_CYCLE.CYCLE_SELECTED_AUX )
      I_Contact( "DB2031_CYCLES_GENERAL".CALIBRATION_CYCLE.CYCLE_SELECTED )
      { S7_GenerateENO := "TRUE" } Move(in := #FC_NUMBER, out1 => "DB440_MACHINE_ALARM_DECODING".GLOBAL_ALARMS_MACHINE.ALARM_DECODING)
      S_Coil( "DB440_MACHINE_ALARM_DECODING".ALARMS_CENTRAL.SEOC_WARNING )
   END_RUNG
   // the same network as SCL:
   // ENO of a box is taken as its EN; it also drops when the box reports an error
   IF NOT (NOT "DB2031_CYCLES_GENERAL".RUN_OUT.CYCLE_COMPLETED) AND NOT "DB2031_CYCLES_GENERAL".MASTER_MEASUREMENT.CYCLE_SELECTED_AUX AND NOT "DB2031_CYCLES_GENERAL".MASTER_MEASUREMENT.CYCLE_SELECTED AND NOT "DB2031_CYCLES_GENERAL".CALIBRATION_CYCLE.CYCLE_SELECTED_AUX AND NOT "DB2031_CYCLES_GENERAL".CALIBRATION_CYCLE.CYCLE_SELECTED THEN
       "DB440_MACHINE_ALARM_DECODING".GLOBAL_ALARMS_MACHINE.ALARM_DECODING := #FC_NUMBER;
       "DB440_MACHINE_ALARM_DECODING".ALARMS_CENTRAL.SEOC_WARNING := TRUE;
   END_IF;
END_REGION

REGION Network 17: WARNINGS
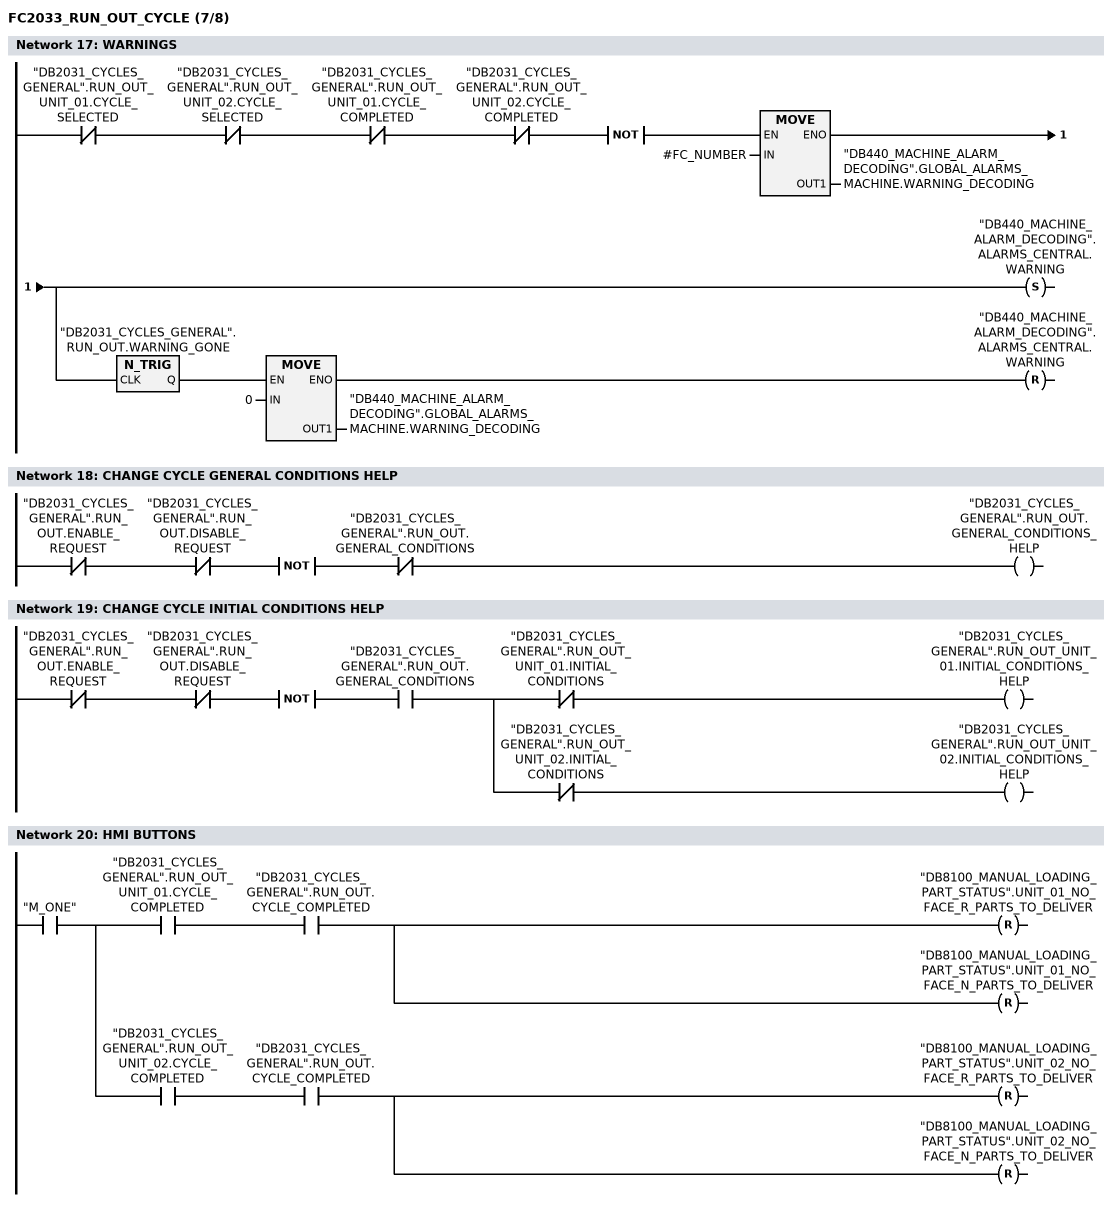
   RUNG wire#powerrail
      I_Contact( "DB2031_CYCLES_GENERAL".RUN_OUT_UNIT_01.CYCLE_SELECTED )
      I_Contact( "DB2031_CYCLES_GENERAL".RUN_OUT_UNIT_02.CYCLE_SELECTED )
      I_Contact( "DB2031_CYCLES_GENERAL".RUN_OUT_UNIT_01.CYCLE_COMPLETED )
      I_Contact( "DB2031_CYCLES_GENERAL".RUN_OUT_UNIT_02.CYCLE_COMPLETED )
      Not()
      Move(in := #FC_NUMBER, out1 => "DB440_MACHINE_ALARM_DECODING".GLOBAL_ALARMS_MACHINE.WARNING_DECODING)
      wire#w1
      S_Coil( "DB440_MACHINE_ALARM_DECODING".ALARMS_CENTRAL.WARNING )
   END_RUNG
   RUNG wire#w1
      N_Trig( "DB2031_CYCLES_GENERAL".RUN_OUT.WARNING_GONE )
      Move(in := 0, out1 => "DB440_MACHINE_ALARM_DECODING".GLOBAL_ALARMS_MACHINE.WARNING_DECODING)
      R_Coil( "DB440_MACHINE_ALARM_DECODING".ALARMS_CENTRAL.WARNING )
   END_RUNG
   // the same network as SCL:
   #_w1 := NOT (NOT "DB2031_CYCLES_GENERAL".RUN_OUT_UNIT_01.CYCLE_SELECTED AND NOT "DB2031_CYCLES_GENERAL".RUN_OUT_UNIT_02.CYCLE_SELECTED AND NOT "DB2031_CYCLES_GENERAL".RUN_OUT_UNIT_01.CYCLE_COMPLETED AND NOT "DB2031_CYCLES_GENERAL".RUN_OUT_UNIT_02.CYCLE_COMPLETED);
   IF #_w1 THEN
       "DB440_MACHINE_ALARM_DECODING".GLOBAL_ALARMS_MACHINE.WARNING_DECODING := #FC_NUMBER;
       "DB440_MACHINE_ALARM_DECODING".ALARMS_CENTRAL.WARNING := TRUE;
   END_IF;
   #_w2 := NOT #_w1 AND "DB2031_CYCLES_GENERAL".RUN_OUT.WARNING_GONE;   // falling edge
   "DB2031_CYCLES_GENERAL".RUN_OUT.WARNING_GONE := #_w1;
   IF #_w2 THEN
       "DB440_MACHINE_ALARM_DECODING".GLOBAL_ALARMS_MACHINE.WARNING_DECODING := 0;
       "DB440_MACHINE_ALARM_DECODING".ALARMS_CENTRAL.WARNING := FALSE;
   END_IF;
END_REGION

REGION Network 18: CHANGE CYCLE GENERAL CONDITIONS HELP
   RUNG wire#powerrail
      I_Contact( "DB2031_CYCLES_GENERAL".RUN_OUT.ENABLE_REQUEST )
      I_Contact( "DB2031_CYCLES_GENERAL".RUN_OUT.DISABLE_REQUEST )
      Not()
      I_Contact( "DB2031_CYCLES_GENERAL".RUN_OUT.GENERAL_CONDITIONS )
      Coil( "DB2031_CYCLES_GENERAL".RUN_OUT.GENERAL_CONDITIONS_HELP )
   END_RUNG
   // the same network as SCL:
   "DB2031_CYCLES_GENERAL".RUN_OUT.GENERAL_CONDITIONS_HELP := NOT (NOT "DB2031_CYCLES_GENERAL".RUN_OUT.ENABLE_REQUEST AND NOT "DB2031_CYCLES_GENERAL".RUN_OUT.DISABLE_REQUEST) AND NOT "DB2031_CYCLES_GENERAL".RUN_OUT.GENERAL_CONDITIONS;
END_REGION

REGION Network 19: CHANGE CYCLE INITIAL CONDITIONS HELP
   RUNG wire#powerrail
      I_Contact( "DB2031_CYCLES_GENERAL".RUN_OUT.ENABLE_REQUEST )
      I_Contact( "DB2031_CYCLES_GENERAL".RUN_OUT.DISABLE_REQUEST )
      Not()
      Contact( "DB2031_CYCLES_GENERAL".RUN_OUT.GENERAL_CONDITIONS )
      wire#w1
      I_Contact( "DB2031_CYCLES_GENERAL".RUN_OUT_UNIT_01.INITIAL_CONDITIONS )
      Coil( "DB2031_CYCLES_GENERAL".RUN_OUT_UNIT_01.INITIAL_CONDITIONS_HELP )
   END_RUNG
   RUNG wire#w1
      I_Contact( "DB2031_CYCLES_GENERAL".RUN_OUT_UNIT_02.INITIAL_CONDITIONS )
      Coil( "DB2031_CYCLES_GENERAL".RUN_OUT_UNIT_02.INITIAL_CONDITIONS_HELP )
   END_RUNG
   // the same network as SCL:
   #_w1 := NOT (NOT "DB2031_CYCLES_GENERAL".RUN_OUT.ENABLE_REQUEST AND NOT "DB2031_CYCLES_GENERAL".RUN_OUT.DISABLE_REQUEST) AND "DB2031_CYCLES_GENERAL".RUN_OUT.GENERAL_CONDITIONS;
   "DB2031_CYCLES_GENERAL".RUN_OUT_UNIT_01.INITIAL_CONDITIONS_HELP := #_w1 AND NOT "DB2031_CYCLES_GENERAL".RUN_OUT_UNIT_01.INITIAL_CONDITIONS;
   "DB2031_CYCLES_GENERAL".RUN_OUT_UNIT_02.INITIAL_CONDITIONS_HELP := #_w1 AND NOT "DB2031_CYCLES_GENERAL".RUN_OUT_UNIT_02.INITIAL_CONDITIONS;
END_REGION

REGION Network 20: HMI BUTTONS
   RUNG wire#powerrail
      Contact( "M_ONE" )
      wire#w1
      Contact( "DB2031_CYCLES_GENERAL".RUN_OUT_UNIT_01.CYCLE_COMPLETED )
      Contact( "DB2031_CYCLES_GENERAL".RUN_OUT.CYCLE_COMPLETED )
      wire#w2
      R_Coil( "DB8100_MANUAL_LOADING_PART_STATUS".UNIT_01_NO_FACE_R_PARTS_TO_DELIVER )
   END_RUNG
   RUNG wire#w2
      R_Coil( "DB8100_MANUAL_LOADING_PART_STATUS".UNIT_01_NO_FACE_N_PARTS_TO_DELIVER )
   END_RUNG
   RUNG wire#w1
      Contact( "DB2031_CYCLES_GENERAL".RUN_OUT_UNIT_02.CYCLE_COMPLETED )
      Contact( "DB2031_CYCLES_GENERAL".RUN_OUT.CYCLE_COMPLETED )
      wire#w3
      R_Coil( "DB8100_MANUAL_LOADING_PART_STATUS".UNIT_02_NO_FACE_R_PARTS_TO_DELIVER )
   END_RUNG
   RUNG wire#w3
      R_Coil( "DB8100_MANUAL_LOADING_PART_STATUS".UNIT_02_NO_FACE_N_PARTS_TO_DELIVER )
   END_RUNG
   // the same network as SCL:
   IF "M_ONE" AND "DB2031_CYCLES_GENERAL".RUN_OUT_UNIT_01.CYCLE_COMPLETED AND "DB2031_CYCLES_GENERAL".RUN_OUT.CYCLE_COMPLETED THEN
       "DB8100_MANUAL_LOADING_PART_STATUS".UNIT_01_NO_FACE_R_PARTS_TO_DELIVER := FALSE;
       "DB8100_MANUAL_LOADING_PART_STATUS".UNIT_01_NO_FACE_N_PARTS_TO_DELIVER := FALSE;
   END_IF;
   IF "M_ONE" AND "DB2031_CYCLES_GENERAL".RUN_OUT_UNIT_02.CYCLE_COMPLETED AND "DB2031_CYCLES_GENERAL".RUN_OUT.CYCLE_COMPLETED THEN
       "DB8100_MANUAL_LOADING_PART_STATUS".UNIT_02_NO_FACE_R_PARTS_TO_DELIVER := FALSE;
       "DB8100_MANUAL_LOADING_PART_STATUS".UNIT_02_NO_FACE_N_PARTS_TO_DELIVER := FALSE;
   END_IF;
END_REGION

REGION Network 21: HMI STATUS
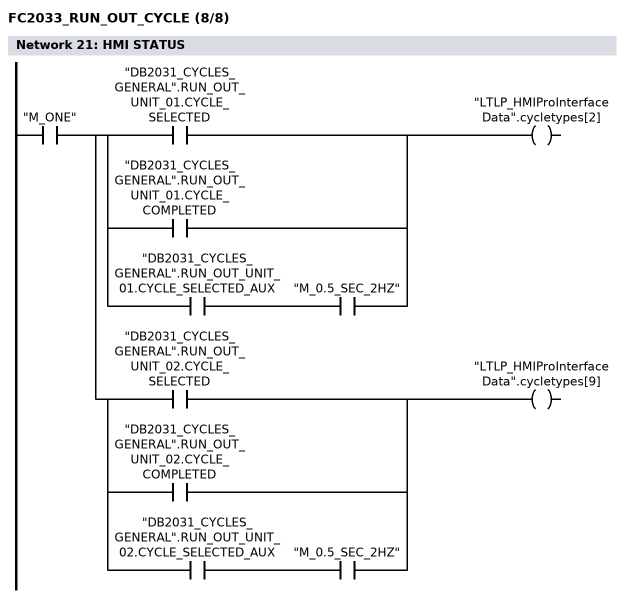
   RUNG wire#powerrail
      Contact( "M_ONE" )
      wire#w1
      Contact( "DB2031_CYCLES_GENERAL".RUN_OUT_UNIT_01.CYCLE_SELECTED )
      wire#w2
      Coil( "LTLP_HMIProInterfaceData".cycletypes[2] )
   END_RUNG
   RUNG wire#w1
      Contact( "DB2031_CYCLES_GENERAL".RUN_OUT_UNIT_01.CYCLE_COMPLETED )
   END_RUNG wire#w2
   RUNG wire#w1
      Contact( "DB2031_CYCLES_GENERAL".RUN_OUT_UNIT_01.CYCLE_SELECTED_AUX )
      Contact( "M_0.5_SEC_2HZ" )
   END_RUNG wire#w2
   RUNG wire#w1
      Contact( "DB2031_CYCLES_GENERAL".RUN_OUT_UNIT_02.CYCLE_SELECTED )
      wire#w3
      Coil( "LTLP_HMIProInterfaceData".cycletypes[9] )
   END_RUNG
   RUNG wire#w1
      Contact( "DB2031_CYCLES_GENERAL".RUN_OUT_UNIT_02.CYCLE_COMPLETED )
   END_RUNG wire#w3
   RUNG wire#w1
      Contact( "DB2031_CYCLES_GENERAL".RUN_OUT_UNIT_02.CYCLE_SELECTED_AUX )
      Contact( "M_0.5_SEC_2HZ" )
   END_RUNG wire#w3
   // the same network as SCL:
   "LTLP_HMIProInterfaceData".cycletypes[2] := "M_ONE" AND ("DB2031_CYCLES_GENERAL".RUN_OUT_UNIT_01.CYCLE_SELECTED OR "DB2031_CYCLES_GENERAL".RUN_OUT_UNIT_01.CYCLE_COMPLETED OR ("DB2031_CYCLES_GENERAL".RUN_OUT_UNIT_01.CYCLE_SELECTED_AUX AND "M_0.5_SEC_2HZ"));
   "LTLP_HMIProInterfaceData".cycletypes[9] := "M_ONE" AND ("DB2031_CYCLES_GENERAL".RUN_OUT_UNIT_02.CYCLE_SELECTED OR "DB2031_CYCLES_GENERAL".RUN_OUT_UNIT_02.CYCLE_COMPLETED OR ("DB2031_CYCLES_GENERAL".RUN_OUT_UNIT_02.CYCLE_SELECTED_AUX AND "M_0.5_SEC_2HZ"));
END_REGION
END_FUNCTION
